FUNCTION F_GetTransportTube : ST_TransportTube
VAR_INPUT
	eTT : T_TransportTube;
END_VAR
VAR
END_VAR

CASE eTT OF
E_InputTransportTube.BI1:
	F_GetTransportTube := GVL_TransportTubes.stBI1;
E_OutputTransportTube.BO4:
	F_GetTransportTube := GVL_TransportTubes.stBO4;
END_CASE

END_FUNCTION

(* stored: Version 1.1.0.1, ProductVersion 3.1.4022.17
   POU F_GetTransportTube: Id {1c225a2d-c668-4975-8e19-7e053353ec27}, SpecialFunc None *)
